(* CODESYS project OOP example __New Operator.project

Project tree, tasks and I/O mapping:
  Device : CODESYS Control for Raspberry Pi SL, 3S - Smart Software Solutions GmbH, version 3.5.12.30
    application Application
      libraries: Standard, * (System); VisuDialogs, * (System); SysFile, 3.5.9.0 (System); AlarmManager, 3.5.12.0 (Intern)
      task MainTask (cyclic, interval 500 ms, priority 1, watchdog 1000 ms x 1) calls New
      program New [ST]
    SoftMotion General Axis Pool
    I²C
    SPI
    GPIOs_A_B : GPIOs B+/Pi2, 3S - Smart Software Solutions GmbH, version 3.5.11.0
        unmapped channels: digital inputs (GPIO0..GPIO31), digital outputs (GPIO0..GPIO31)
    Onewire
    Camera device
      <Empty>
  libraries: VisuSymbols, 3.5.10.0 (System)
  New/
    function block FB_Dynamic [ST]
    data type myDUT
*)

// New/myDUT
{attribute 'enable_dynamic_creation'}
TYPE myDUT :
    STRUCT
     a,b,c,d,e,f : INT;
    END_STRUCT
END_TYPE

// Device/Application/New
(* 
	This operator is an extension of the IEC 61131-3 standard.
	The __NEW operator reserves memory for function block instances or arrays of standard data types. 
	The operator returns a matching typed pointer to the object. 
	If you do not use the operator within an assignment, then CODESYS prints an error message.
	If the attempt to allocate memory fails, then __NEW returns the value 0.
	
		* Requirement: In the properties dialog of the application, the Use dynamic memory allocation check box is selected in the Application build options tab.
	
	=> APPLICATION / PROPERTIES / TAB APPLICATION BUILD OPTIONS / SET "Use dynamic memory allocation check box", SET "Memory Usage (1024KB)"
	
	
 	NOTICE! 
		A function block that can be created with __NEW has a fixed memory area. 
		It cannot modify its data layout by means of an online change. 
		Therefore, new variables cannot be added or deleted, and types cannot be modified. 
		This makes sure that the pointer to this object is also valid after an online change.
 
		For this reason, the __NEW operator can be applied only to function blocks from libraries and function blocks 
		with the attribute "enable_dynamic_creation". If the interface of this kind of function block is changed, then CODESYS issues an error message.

	NOTICE! 
		Two tasks should not call __NEW at the same time. 
		Either you use a semaphore (SysSemEnter) or comparable method to prevent any concurrent calling of __NEW, 
		or you use __NEW in one tasks only (recommended).
 
*)

PROGRAM New
VAR
	pDut : POINTER TO myDUT;
	xInit : BOOL := TRUE;
	bDelete : BOOL;
	pFB : POINTER TO FB_Dynamic;
	loc : INT;
	pArrayBytes : POINTER TO BYTE;
	test : INT;
	parr : POINTER TO BYTE;
END_VAR

IF (xInit) THEN
    pDut := __NEW(myDUT);
	pFB := __NEW(FB_Dynamic);
	pArrayBytes := __NEW(BYTE, 25);
    xInit := FALSE;
END_IF

IF pDut <> 0 THEN
	pDut^.a := pDut^.f + 1;
	pDut^.b := pDut^.a + 1;
	pDut^.c := pDut^.b + 1;
	pDut^.d := pDut^.c + 1;
	pDut^.e := pDut^.d + 1;
	pDut^.f := pDut^.e + 1;
END_IF

IF pFB <> 0 THEN
	pFB^();				// call fb
END_IF

IF (bDelete) THEN
	__DELETE(pDut); 
	__DELETE(pFB); 
	__DELETE(pArrayBytes);
END_IF

END_PROGRAM

// New/FB_Dynamic
{attribute 'enable_dynamic_creation'} // Mandatory
FUNCTION_BLOCK FB_Dynamic
VAR_INPUT
    in1 : INT;
	in2 : INT;
END_VAR
VAR_OUTPUT
    out : INT;
END_VAR

out := in1 + in2;

END_FUNCTION_BLOCK
